// Mitsubishi GX Works2 project: 0624(인터록회로_다중스위치)   PLC: Q02/Q02H

PROGRAM MAIN
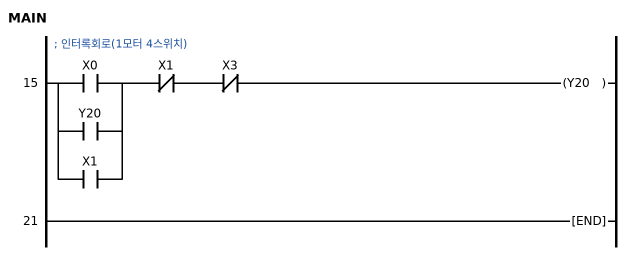
; 인터록회로(1모터 4스위치)
15    LD      X0
      OR      Y20
      OR      X1
      ANI     X1
      ANI     X3
      OUT     Y20
21    END
END_PROGRAM
